// TwinCAT 3 PLC project PLC
// ProgramVersion: 3.1.4023.0
// libraries:
//   Tc2_Standard, * (Beckhoff Automation GmbH)
//   Tc2_System, * (Beckhoff Automation GmbH)
//   Tc2_Utilities, * (Beckhoff Automation GmbH)
//   Tc3_Module, * (Beckhoff Automation GmbH)
//   VisuDialogs, * (System)
//   VisuSymbols,3.5.10.0,System
// project tree:
//   / GlobalTextList.TcGTLO, PlcTask.TcTTO, Visualization Manager.TcVMO (not stored)
//   GVLs/ GVL_Elementy.TcGVL, GVL_Wejscia_IO.TcGVL, GVL_Wyjscia_IO.TcGVL (not stored)
//   POUs/01 - Elementy/Czujnik/ITF/ ITF_Czujnik.TcIO (not stored)
//   POUs/01 - Elementy/Czujnik/POU/ FB_Czujnik_NO.TcPOU (not stored), FB_Czujnik_NC.TcPOU (not stored)
//   POUs/01 - Elementy/Elektrozawór/ITF/ ITF_Elektozawor.TcIO (not stored)
//   POUs/01 - Elementy/Elektrozawór/POU/ FB_Elektrozawor_5na2_1Cewka.TcPOU (not stored), FB_Elektrozawor_5na2_2Cewki.TcPOU (not stored), FB_Elektrozawor_5na3_Odpowietrzony.TcPOU (not stored), FB_Elektrozawor_5na3_Zapowietrzony.TcPOU (not stored)
//   POUs/01 - Elementy/Silownik/DUT/ DUT_SilownikParametry.TcDUT (not stored)
//   POUs/01 - Elementy/Silownik/ITF/ ITF_Silownik.TcIO (not stored)
//   POUs/01 - Elementy/Silownik/POU/ FB_Silownik.TcPOU (not stored), FB_Silownik_Kontola.TcPOU (not stored), FB_Silownik_Kontrola_Komunikacja.TcPOU (not stored)
//   POUs/02 -Przesuwacz Na Silowniku/DUT/ DUT_PrzesuwaczNaSilowniku_Parametry.TcDUT (not stored)
//   POUs/02 -Przesuwacz Na Silowniku/POU/ FB_PrzesuwaczNaSilowniku.TcPOU, FB_PrzesuwaczNaSilowniku_Komunikacja.TcPOU (not stored)
//   POUs/10 - Logowanie błędów/DUT/ DUT_LogowanieBledow_Zapamietanych.TcDUT (not stored), DUT_LogowanieBledow_ZdarzenieOpis.TcDUT (not stored), DUT_LogowanieBledow_Zdarzenie.TcDUT (not stored), DUT_LogowanieBledow_ZdarzenieStan.TcDUT (not stored), DUT_LogowanieBledow_ZdarzenieWyswietlane.TcDUT, DUT_LogowanieBledow_WyswietlanieParametry.TcDUT (not stored)
//   POUs/10 - Logowanie błędów/GVL/ GVL_LogowanieBledow.TcGVL, GVL_LogowanieBledow_Stale.TcGVL
//   POUs/10 - Logowanie błędów/ITF/ ITF_LogowanieBledow_ElementWykonawczy.TcIO (not stored)
//   POUs/10 - Logowanie błędów/POU/ FB_LogowanieBledow.TcPOU, FB_LogowanieBledow_ElementWykonawczy.TcPOU, FB_LogowanieBledow_ElementZlozony.TcPOU
//   POUs/10 - Logowanie błędów/Wizualizacja/ Visu_LogowanieBledow_Tabela.TcVIS
//   POUs/ MAIN.TcPOU
//   VISUs/ Visualization.TcVIS
// real-time tasks:
//   TASK PlcTask: cycle T#10ms, priority 20, ADS port 350

CONFIGURATION PLC
    RESOURCE PLC ON TwinCAT3
        TASK PlcTask(INTERVAL := T#10ms, PRIORITY := 20);
        PROGRAM MAIN WITH PlcTask : MAIN;
    END_RESOURCE
END_CONFIGURATION

// ---- POUs/10 - Logowanie błędów/DUT/DUT_LogowanieBledow_ZdarzenieWyswietlane.TcDUT
TYPE DUT_LogowanieBledow_ZdarzenieWyswietlane :
STRUCT
	sNrKomponentu							: STRING[10];
	sKodBledu								: STRING[10];
	byRodzajZdarzenia						: BYTE;
	sOpis									: STRING;
	dtDataStart								: DT;
	dtDateKoniec							: DT;
	dwKolor									: UDINT;
END_STRUCT
END_TYPE

// ---- GVLs/GVL_Elementy.TcGVL
{attribute 'qualified_only'}
{attribute 'global_init_slot' := '40520'}
VAR_GLOBAL
	fbSilownik								: FB_Silownik_Kontola (		fbCzujnikPozycja0 			:= GVL_Wejscia_IO.bCzujnik0S1, 
																		fbCzujnikPozycjaMax 		:= GVL_Wejscia_IO.bCzujnikMaxS1,
																		fbElektrozawor 				:= GVL_Wyjscia_IO.fbElektrozaworS1);
	fbSilownik1								: FB_Silownik_Kontola (		fbCzujnikPozycja0 			:= GVL_Wejscia_IO.bCzujnik0S2, 
																		fbCzujnikPozycjaMax 		:= GVL_Wejscia_IO.bCzujnikMaxS2,
																		fbElektrozawor 				:= GVL_Wyjscia_IO.fbElektrozaworS2);																
	fbPrzesuwacz							: FB_PrzesuwaczNaSilowniku (bCzujnik0Zabieraka			:= GVL_Wejscia_IO.bCzujnik0Z,
		                                                                bCzujnikMaxZabieraka		:= GVL_Wejscia_IO.bCzujnikMaxZ	,
	                                                                    fbElektrozaworZabieraka		:= GVL_Wyjscia_IO.fbElektrozaworZ,
	                                                                    bCzujnik0Przesuwacza		:= GVL_Wejscia_IO.bCzujnik0P,
	                                                                    bCzujnikMaxPrzesuwacza		:= GVL_Wejscia_IO.bCzujnikMaxP	,
	                                                                    fbElektrozaworPrzesuwacza	:= GVL_Wyjscia_IO.fbElektrozaworP);
END_VAR

// ---- GVLs/GVL_Wejscia_IO.TcGVL
{attribute 'qualified_only'}
{attribute 'global_init_slot' := '40501'}
VAR_GLOBAL
//czujniki siłownik1
	bCzujnik0S1								: FB_Czujnik_NO;
	bCzujnikMaxS1							: FB_Czujnik_NO;
//czujniki siłownika2 
	bCzujnik0S2								: FB_Czujnik_NO;
	bCzujnikMaxS2							: FB_Czujnik_NO;
//czujniki przesuwacza
	bCzujnik0Z								: FB_Czujnik_NO;
	bCzujnikMaxZ							: FB_Czujnik_NO;
	bCzujnik0P								: FB_Czujnik_NO;
	bCzujnikMaxP							: FB_Czujnik_NO;
END_VAR

// ---- POUs/10 - Logowanie błędów/GVL/GVL_LogowanieBledow.TcGVL
{attribute 'qualified_only'}
{attribute 'global_init_slot' := '40550'}
VAR_GLOBAL
	arrElementyWykonawcze 					: ARRAY [1..GVL_LogowanieBledow_Stale.MAX_ILOSC_ELEMENTOW] OF 
																ITF_LogowanieBledow_ElementWykonawczy := [
																	GVL_Elementy.fbSilownik.fbLBKomunikacja, 
																	GVL_Elementy.fbSilownik1.fbLBKomunikacja,
																	GVL_Elementy.fbPrzesuwacz.fbLBKomunikacja];

	fbLoger 								: FB_LogowanieBledow (	tablica := arrElementyWykonawcze,
																	iIloscDodanychElementow := 3);
																	
	
END_VAR
VAR_GLOBAL //PERSISTENT
	arrTablicaZdarzenZapamietancyh			: ARRAY [1..GVL_LogowanieBledow_Stale.MAX_ILOSC_ZDARZEN_ZAPAMIETANYCH] OF DUT_LogowanieBledow_Zapamietanych;																
	
	iIloscZdarzenZapamietanych				: INT;	//ilosc zdarzen ktore wystapiły
END_VAR

// ---- POUs/10 - Logowanie błędów/GVL/GVL_LogowanieBledow_Stale.TcGVL
{attribute 'qualified_only'}
VAR_GLOBAL CONSTANT
	MAX_ILOSC_ELEMENTOW						: INT := 10; //Ilementów głównych
	MAX_ILOSC_ZDARZEN_NA_ELEMENT			: INT := 10;
	MAX_ILOSC_ELEMENTOW_NA_PODZESPOL		: INT := 10;
	MAX_ILOSC_ZDARZEN						: INT := 100;
	MAX_ILOSC_ZDARZEN_DO_WYSWIETLANIA		: INT := 50;
END_VAR

// ---- POUs/MAIN.TcPOU
//==================================================================================================
//								RJM Maszyny sp. z o.o.
//									13.05.2022
//	Program główny sterujący  
// 	v1.0	|| TC v 3.1.4024.29		|| - pierwsza wersja
//==================================================================================================
PROGRAM MAIN
VAR
	bDoPoczatku								: BOOL;
	bDoKonca								: BOOL;
	bNaPoczatku								: BOOL;
	bNaKoncu								: BOOL;
	bWykonajCyklPrzesuwania					: BOOL;
	bWyswietlAlarmy							: BOOL;

END_VAR

(* 	DO ZROBIENIA
	LOGOWANIE BLEDOW
		- poprawić wizualizację logowania błędów nie działają przyciski wyboru rodzaju informacji 
		- id zdarzenia to string nei da się filtrować po id bo nei da się wpisać numerka
		- na maszynie odznaczyc PERSISTENT
		- funkcja czyszczenia tablicy zapamietanych 
	
*)

//--------TESTY FB SILOWNIK
	GVL_Elementy.fbSilownik.Praca ();
	GVL_Elementy.fbPrzesuwacz.Praca ();
	
	IF (bDoPoczatku) THEN
		GVL_Elementy.fbSilownik.PrzesunDoPoczatku	:= TRUE;
		bDoPoczatku							:= FALSE;
	END_IF
	
	IF (bDoKonca) THEN
		GVL_Elementy.fbSilownik.PrzesunDoKonca	:= TRUE;
		bDoKonca							:= FALSE;
	END_IF
	
	bNaPoczatku								:= GVL_Elementy.fbSilownik.NaPoczatku;
	bNaKoncu								:= GVL_Elementy.fbSilownik.NaKoncu;
	
	IF (bWykonajCyklPrzesuwania) THEN
		GVL_Elementy.fbPrzesuwacz.WykonajCyklPrzesuwania	:= TRUE;
		bWykonajCyklPrzesuwania				:= FALSE;
	END_IF
//--------TESTY FB SILOWNIK
//--------LOGER
	GVL_LogowanieBledow.fbLoger (arrZdarzeniaPamietane 		:= GVL_LogowanieBledow.arrTablicaZdarzenZapamietancyh,
								iIloscZdarzenZapamietanych 	:= GVL_LogowanieBledow.iIloscZdarzenZapamietanych,
								bWyswietlanieTablicyAlarmow	:= bWyswietlAlarmy);
//--------LOGER
												
//--------STEROWANIE MASZYNĄ

//--------STEROWANIE MASZYNĄ

END_PROGRAM

// ---- POUs/02 -Przesuwacz Na Silowniku/POU/FB_PrzesuwaczNaSilowniku.TcPOU
//==================================================================================================
//								RJM Maszyny sp. z o.o.
//									13.05.2022
//	Obsluga przesuwacza na siłowniku 
//	Siłownik zabieraka plus siłownik przesuwający 
//	Cykl przesuwania: wysun zabierak -> przesun -> schowaj zabierak -> powrót  
// 	v1.0	|| TC v 3.1.4024.22		|| - pierwsza wersja
//==================================================================================================
FUNCTION_BLOCK FB_PrzesuwaczNaSilowniku
VAR_INPUT
END_VAR
VAR_OUTPUT
END_VAR
VAR
	bCzujnik0Zabieraka						: ITF_Czujnik;
	bCzujnikMaxZabieraka					: ITF_Czujnik;
	fbElektrozaworZabieraka					: ITF_Elektozawor;
	bCzujnik0Przesuwacza					: ITF_Czujnik;
	bCzujnikMaxPrzesuwacza					: ITF_Czujnik;
	fbElektrozaworPrzesuwacza				: ITF_Elektozawor;
	fbZabierak								: FB_Silownik_Kontola (fbCzujnikPozycja0 		:= bCzujnik0Zabieraka, 
																	fbCzujnikPozycjaMax 	:= bCzujnikMaxZabieraka,
																	fbElektrozawor 			:= fbElektrozaworZabieraka);
	fbPrzesuwaczNaped						: FB_Silownik_Kontola (fbCzujnikPozycja0 		:= bCzujnik0Przesuwacza, 
																	fbCzujnikPozycjaMax 	:= bCzujnikMaxPrzesuwacza,
																	fbElektrozawor 			:= fbElektrozaworPrzesuwacza);	
	arrElementyWykonawcze 					: ARRAY [1..10] OF ITF_LogowanieBledow_ElementWykonawczy := 
														[fbZabierak.fbLBKomunikacja, 
														fbPrzesuwaczNaped.fbLBKomunikacja];
	fbLBKomunikacja							: FB_PrzesuwaczNaSilowniku_Komunikacja 
														(arrElementyWykonawcze := arrElementyWykonawcze,
														iIloscPodlementow := 2);
END_VAR

METHOD FB_init : BOOL
VAR_INPUT
	bInitRetains : BOOL; // if TRUE, the retain variables are initialized (warm start / cold start)
	bInCopyCode : BOOL;  // if TRUE, the instance afterwards gets moved into the copy code (online change)
	bCzujnik0Zabieraka						: ITF_Czujnik;
	bCzujnikMaxZabieraka					: ITF_Czujnik;
	fbElektrozaworZabieraka					: ITF_Elektozawor;
	bCzujnik0Przesuwacza					: ITF_Czujnik;
	bCzujnikMaxPrzesuwacza					: ITF_Czujnik;
	fbElektrozaworPrzesuwacza				: ITF_Elektozawor;
END_VAR
THIS^.bCzujnik0Zabieraka					:= bCzujnik0Zabieraka;			     
THIS^.bCzujnikMaxZabieraka					:= bCzujnikMaxZabieraka;		    
THIS^.fbElektrozaworZabieraka				:= fbElektrozaworZabieraka;		 
THIS^.bCzujnik0Przesuwacza					:= bCzujnik0Przesuwacza;		    
THIS^.bCzujnikMaxPrzesuwacza				:= bCzujnikMaxPrzesuwacza;		  
THIS^.fbElektrozaworPrzesuwacza				:= fbElektrozaworPrzesuwacza;

THIS^.fbZabierak.FB_init (FALSE, FALSE, bCzujnik0Zabieraka, bCzujnikMaxZabieraka, fbElektrozaworZabieraka);
THIS^.fbPrzesuwaczNaped.FB_init (FALSE, FALSE, bCzujnik0Przesuwacza, bCzujnikMaxPrzesuwacza, fbElektrozaworPrzesuwacza);
END_METHOD

END_FUNCTION_BLOCK

// ---- POUs/10 - Logowanie błędów/POU/FB_LogowanieBledow.TcPOU
//==================================================================================================
//							RJM MASZYNY SP. Z O>O>
//									05.02.2022
//	Metoda sterujaca logowaniem bledow
// 	v1.0	|| TC v 3.1.4024.22		|| - pierwsza wersja
//==================================================================================================
FUNCTION_BLOCK FB_LogowanieBledow
VAR_INPUT
	arrZdarzeniaPamietane					: REFERENCE TO ARRAY [1..GVL_LogowanieBledow_Stale.MAX_ILOSC_ZDARZEN_ZAPAMIETANYCH] OF DUT_LogowanieBledow_Zapamietanych;
	iIloscZdarzenZapamietanych				: REFERENCE TO INT;
	bWyswietlanieTablicyAlarmow				: BOOL;
END_VAR
VAR_OUTPUT
END_VAR
VAR
	arrTablicaElementowWykonawczych 		: ARRAY [1..GVL_LogowanieBledow_Stale.MAX_ILOSC_ELEMENTOW] OF ITF_LogowanieBledow_ElementWykonawczy;
	iIloscDodanychElementow					: INT;			//ilość dodanych elementow wykonawczych, przypisać w deklaracji
	iIloscDodanychWszystkichZdarzen 		: INT;			//ilosść dodanych zdarzeń globalnie
	iJezykID								: INT := 1045;	//id języka - domyślnie polski
	bwypelnij								: BOOL;			//Wypełnienie tablic - wykonać na początku i po zmianie języka
	bDaneWypelnione							: BOOL := FALSE;//jak true mozna odczytywac stany podzespolow
	iI										: INT;
	iJ										: INT;
	
	arrTablicaDefinicjiZdarzen				: ARRAY [1..GVL_LogowanieBledow_Stale.MAX_ILOSC_ZDARZEN] OF DUT_LogowanieBledow_Zdarzenie;
	arrTablicaDefinicjiZdarzenOpis			: ARRAY [1..GVL_LogowanieBledow_Stale.MAX_ILOSC_ZDARZEN] OF DUT_LogowanieBledow_ZdarzenieOpis;
	arrTablicaDefinicjiZdarzenStan			: ARRAY [1..GVL_LogowanieBledow_Stale.MAX_ILOSC_ZDARZEN] OF DUT_LogowanieBledow_ZdarzenieStan;
	arrTablicaWyswietlana					: ARRAY [1..GVL_LOgowanieBledow_Stale.MAX_ILOSC_ZDARZEN_DO_WYSWIETLANIA] OF DUT_LogowanieBledow_ZdarzenieWyswietlane;
	arrPoczatekZdarzenia					: ARRAY [1..GVL_LogowanieBledow_Stale.MAX_ILOSC_ZDARZEN] OF R_TRIG;
	arrKoniecZdarzenia						: ARRAY [1..GVL_LogowanieBledow_Stale.MAX_ILOSC_ZDARZEN] OF F_TRIG;

	fbLocalSystemTime						: FB_LocalSystemTime;
	stAktualnyCzas							: TIMESTRUCT;				// Aktualny czas sytemowy w formie struktury
	dtAktualnyCzas							: DT;		
	bBladRozmiaruTablicyMozliwychZdarzen	: BOOL;						// Niewlasciwy rozmiar tablicy zdarzen - sprawdz HS_ILOSC_ZDARZEN_PAMIETANYCH
	bReferencjaOK							: BOOL;
	bInicjalizacjaDanychTablicyPamietanych	: BOOL := FALSE;
	tonOdswierzanieTablicyPamieci			: TON;
	tOdswierzenieTablicyPamieci				: TIME := T#100MS;
	bOdswierzanieCiagle						: BOOL;
	tonOdswierzaniaTablicyWyswietlania		: TON;
	tOdswierzaniaTablicyWyswietlania		: TIME := T#200MS;
	stWyswietlanieParametry					: DUT_LogowanieBledow_WyswietlanieParametry;
	bWiecejDanychZapamietanych				: BOOL;	//informacja ze jest wiecej danych zapamietanych niz do wyswietlenia
END_VAR

//Pobranie aktualnego czasu systemu
	fbLocalSystemTime (bEnable:= TRUE, systemTime=> stAktualnyCzas);
	dtAktualnyCzas								:= SYSTEMTIME_TO_DT(stAktualnyCzas);
//Sprawdzenie błędów rozmiaru tablic 
	bBladRozmiaruTablicyMozliwychZdarzen 		:= GVL_LogowanieBledow_Stale.MAX_ILOSC_ZDARZEN < 5 OR
													GVL_LogowanieBledow_Stale.MAX_ILOSC_ZDARZEN > 1000;
//Nie ma błędów pracuj z tablicami
	bReferencjaOK := __ISVALIDREF (arrZdarzeniaPamietane);

	IF (NOT bBladRozmiaruTablicyMozliwychZdarzen AND bReferencjaOK) THEN
	//Inicjalizacja tablicy przy starcie 
		Inicjalizacja ();
	//Wypełnienie tablicy zdarzen dla wszystkich elementow
		IF(bwypelnij) THEN
			WypelnianieTablicyZdarzen ();
		END_IF
	//Aktualizacja tablicy stanów
	//Timer odswiezania
		tonOdswierzanieTablicyPamieci(IN:= NOT tonOdswierzanieTablicyPamieci.Q, PT:= tOdswierzenieTablicyPamieci, Q=> , ET=> );
		IF (bDaneWypelnione AND (bOdswierzanieCiagle OR tonOdswierzanieTablicyPamieci.Q)) THEN
			ObslugaAktywnychZdarzen ();
		END_IF		
	//Odswierzanie tablicy alarmow
		tonOdswierzaniaTablicyWyswietlania(IN:= NOT tonOdswierzaniaTablicyWyswietlania.Q,
											 PT:= tOdswierzaniaTablicyWyswietlania, Q=> , ET=> );		// Timer odswiezania
		IF (bWyswietlanieTablicyAlarmow) THEN
			Wyswietlanie ();
		END_IF
	END_IF

METHOD FB_init : BOOL
VAR_INPUT
	bInitRetains : BOOL; // if TRUE, the retain variables are initialized (warm start / cold start)
	bInCopyCode : BOOL;  // if TRUE, the instance afterwards gets moved into the copy code (online change)
	tablica 								: ARRAY [1..GVL_LogowanieBledow_Stale.MAX_ILOSC_ELEMENTOW] OF ITF_LogowanieBledow_ElementWykonawczy;
	iIloscDodanychElementow					: INT;
END_VAR
THIS^.arrTablicaElementowWykonawczych 								:= tablica;
THIS^.iIloscDodanychElementow				:= iIloscDodanychElementow;
END_METHOD

//==================================================================================================
//							RJM MASZYNY SP. Z O>O>
//									05.02.2022
//	Inicjalizacja tablicy zapamietanych zdarzen
//	Wyszukanie niezakonczonych i konczymy
// 	v1.0	|| TC v 3.1.4024.22		|| - pierwsza wersja
//==================================================================================================
METHOD PRIVATE Inicjalizacja : BOOL
VAR_INPUT
END_VAR
		IF (NOT bInicjalizacjaDanychTablicyPamietanych) THEN
			bInicjalizacjaDanychTablicyPamietanych	:= TRUE;
			FOR iJ := 1 TO iIloscZdarzenZapamietanych DO
				IF (arrZdarzeniaPamietane [iJ].bAktywne) THEN
					arrZdarzeniaPamietane [iJ].bAktywne	:= FALSE;
					//wywolac ZadanieKonie();
				END_IF
			END_FOR
		END_IF
END_METHOD

//==================================================================================================
//							RJM MASZYNY SP. Z O>O>
//									05.02.2022
//	Skanowanie tablicy stanow i po pojawieniu sie aktywnego zdarzenia dodajemy do tablicy pamietanych
//	po zakonczeniu aktywnosci zgloszenia zmieniamy w tablicy pamietanych
// 	v1.0	|| TC v 3.1.4024.22		|| - pierwsza wersja
//==================================================================================================
METHOD PRIVATE ObslugaAktywnychZdarzen : BOOL
VAR_INPUT
END_VAR
	FOR iJ := 1 TO iIloscDodanychElementow DO
		arrTablicaElementowWykonawczych [iJ].ZwrocTabliceStanu (arrTablicaDefinicjiZdarzenStan := arrTablicaDefinicjiZdarzenStan);
	END_FOR
	
	FOR iJ := 1 TO iIloscDodanychWszystkichZdarzen DO
		arrPoczatekZdarzenia [iJ] (CLK := arrTablicaDefinicjiZdarzenStan [iJ].bAktywne);
		IF (arrPoczatekZdarzenia [iJ].Q) THEN
		//dodac nowe zdarzenie do tablicy arrZdarzeniaPamietane
			ZdarzeniePoczatek (iIdZdarzenia 	:= arrTablicaDefinicjiZdarzen [iJ].iIdZdarzenia,
								dtAktualnyCzas 	:= dtAktualnyCzas);
		END_IF
		arrKoniecZdarzenia [iJ] (CLK := arrTablicaDefinicjiZdarzenStan [iJ].bAktywne);
		IF (arrKoniecZdarzenia [iJ].Q) THEN
		//odznaczyc koniec zdarzenia w tablicy arrZdarzeniaPamietane
			ZdarzenieKoniec (iNumerWiersza 		:= ZnajdzZdarzenieWTablicyPamietanychPoID (iIDZdarzenia := arrTablicaDefinicjiZdarzen [iJ].iIdZdarzenia),
								dtAktualnyCzas 	:= dtAktualnyCzas);
		END_IF
	END_FOR
END_METHOD

//==================================================================================================
//							RJM MASZYNY SP. Z O>O>
//									05.02.2022
//	Pobieranie danych zdarzen od podelementow systemu i dopisywanie ich do tablicy zdarzen
// 	v1.0	|| TC v 3.1.4024.22		|| - pierwsza wersja
//==================================================================================================
METHOD PRIVATE WypelnianieTablicyZdarzen : BOOL
VAR_INPUT
END_VAR
	bDaneWypelnione						:= FALSE;
	FOR iI := 1 TO iIloscDodanychElementow DO 
		arrTablicaElementowWykonawczych [iI].ZwrocTabliceDefinicji (	
												arrTablicaDefinicjiZdarzen := arrTablicaDefinicjiZdarzen,
												arrTablicaDefinicjiZdarzenOpis := arrTablicaDefinicjiZdarzenOpis,
												arrTablicaDefinicjiZdarzenStan := arrTablicaDefinicjiZdarzenStan,
												iIdZdarzenia := iIloscDodanychWszystkichZdarzen, 
												iNrPodzespolu := iI, 
												iNrPodelementu := 1,
												iNrElementu := 1, 
												iJezykId := iJezykID);
	END_FOR
	bwypelnij 							:= FALSE;
	bDaneWypelnione						:= TRUE;
END_METHOD

//==================================================================================================
//							RJM MASZYNY SP. Z O>O>
//									05.02.2022
//	Start wypelniania tablicy zdarzen
// 	v1.0	|| TC v 3.1.4024.22		|| - pierwsza wersja
//==================================================================================================
PROPERTY WypelnijTabliceZdarzen : BOOL
SET
bwypelnij									:= WypelnijTabliceZdarzen;
END_SET
END_PROPERTY

METHOD PRIVATE Wyswietlanie : BOOL
VAR_INPUT
END_VAR

VAR
	j										: INT;
	i										: INT;
	bUsunZWyswietlania						: BOOL;
END_VAR
IF (tonOdswierzaniaTablicyWyswietlania.Q) THEN
	MEMSET(ADR(arrTablicaWyswietlana),0,SIZEOF(arrTablicaWyswietlana));
	j										:= 1; //wskaznik wierszy tablicy wyswietlania
	bWiecejDanychZapamietanych				:= FALSE;
	FOR i := 1 TO iIloscZdarzenZapamietanych DO
		bUsunZWyswietlania					:= FALSE;	
		IF (arrZdarzeniaPamietane [i].iIDZdarzenia <> 0) THEN	//sprawdzenie czy w wierszu sa jakies dane
			//Ustawienie filtrow wyswietlania
			bUsunZWyswietlania				:= stWyswietlanieParametry.bFiltrID AND stWyswietlanieParametry.iFiltrID <> arrTablicaDefinicjiZdarzen [arrZdarzeniaPamietane [i].iIDZdarzenia].byRodzajZdarzenia;
//			bUsunZWyswietlania				:= bUsunZWyswietlania OR (stWyswietlanieParametry.bFiltrRodzaj AND stWyswietlanieParametry.byFiltrRodzaj <> arrTablicaDefinicjiZdarzen [arrZdarzeniaPamietane [i].iIDZdarzenia].byRodzajZdarzenia);
			bUsunZWyswietlania				:= bUsunZWyswietlania OR (stWyswietlanieParametry.bFiltrStartOD AND arrZdarzeniaPamietane [i].dtDataStart <= stWyswietlanieParametry.dtFiltrStartOD);
			bUsunZWyswietlania				:= bUsunZWyswietlania OR (stWyswietlanieParametry.bFiltrStartDO AND arrZdarzeniaPamietane [i].dtDataStart >= stWyswietlanieParametry.dtFiltrStartDO);
			bUsunZWyswietlania				:= bUsunZWyswietlania OR (stWyswietlanieParametry.bFiltrKoniecOD AND arrZdarzeniaPamietane [i].dtDataKoniec <= stWyswietlanieParametry.dtFiltrKoniecOD);
			bUsunZWyswietlania				:= bUsunZWyswietlania OR (stWyswietlanieParametry.bFiltrKoniecDO AND arrZdarzeniaPamietane [i].dtDataKoniec >= stWyswietlanieParametry.dtFiltrKoniecDO);
			bUsunZWyswietlania				:= bUsunZWyswietlania OR (stWyswietlanieParametry.bFiltrAktywne AND DT#1970-1-1-0:0:0 <> arrZdarzeniaPamietane[i].dtDataKoniec);
			// Analogicznie dodajemy inne filtry jesli jest taka potrzeba
			// Jesli element nie zostal usuniety przez filtr to dodajemy go do tablicy alarmow wyswietlanych
			IF (NOT bUsunZWyswietlania) THEN
				arrTablicaWyswietlana [j].sNrKomponentu	:= arrTablicaDefinicjiZdarzen [i].sNrKomponentu;
				arrTablicaWyswietlana [j].byRodzajZdarzenia	:= arrTablicaDefinicjiZdarzen [i].byRodzajZdarzenia;
 				arrTablicaWyswietlana [j].sOpis			:= arrTablicaDefinicjiZdarzenOpis [i].sOpis;
				arrTablicaWyswietlana [j].sKodBledu		:= arrTablicaDefinicjiZdarzen [i].sKodBledu;
				arrTablicaWyswietlana [j].dtDataStart	:= arrZdarzeniaPamietane [i].dtDataStart;
				arrTablicaWyswietlana [j].dtDataKoniec	:= arrZdarzeniaPamietane [i].dtDataKoniec;
				CASE arrTablicaWyswietlana [j].byRodzajZdarzenia OF
					1	: arrTablicaWyswietlana [j].dwKolor	:= 16#FFFF0000;	// blad 		- czerwony
					2	: arrTablicaWyswietlana [j].dwKolor	:= 16#FFFFFF00;	// ostzrezenie 	- zolty
					3	: arrTablicaWyswietlana [j].dwKolor	:= 16#FFFFFFFF;	// wiadomosc 	- bialy
					4	: arrTablicaWyswietlana [j].dwKolor	:= 16#FF0000FF; // safety 		- niebieski
				END_CASE
				j := j + 1;
			END_IF
		END_IF
		IF (j > GVL_LogowanieBledow_Stale.MAX_ILOSC_ZDARZEN_DO_WYSWIETLANIA) THEN
			bWiecejDanychZapamietanych		:= TRUE;
			EXIT;
		END_IF
	END_FOR
END_IF
END_METHOD

//==================================================================================================
//							RJM MASZYNY SP. Z O>O>
//									05.02.2022
//	Zdarzenie przestalo byc aktywne zmien dane
// 	v1.0	|| TC v 3.1.4024.22		|| - pierwsza wersja
//==================================================================================================
METHOD PRIVATE ZdarzenieKoniec : BOOL
VAR_INPUT
	iNumerWiersza							: INT;	//numer wiersza dla konkretnego IDzdarzenia
	dtAktualnyCzas							: DT;
END_VAR
arrZdarzeniaPamietane [iNumerWiersza].dtDataKoniec	:= dtAktualnyCzas;
arrZdarzeniaPamietane [iNumerWiersza].bAktywne		:= FALSE;
END_METHOD

//==================================================================================================
//							RJM MASZYNY SP. Z O>O>
//									05.02.2022
//	Dodanie nowego aktywnego zdarzenia do tablicy pamietanych
// 	v1.0	|| TC v 3.1.4024.22		|| - pierwsza wersja
//==================================================================================================
METHOD PRIVATE ZdarzeniePoczatek : BOOL
VAR_INPUT
	iIdZdarzenia							: INT;
	dtAktualnyCzas							: DT;
END_VAR
VAR
	i										: INT;
END_VAR
iIloscZdarzenZapamietanych					:= iIloscZdarzenZapamietanych + 1;
// Przesun elemety tablicy
FOR i := 0 TO iIloscZdarzenZapamietanych - 2 DO
	arrZdarzeniaPamietane [iIloscZdarzenZapamietanych - i]	:= arrZdarzeniaPamietane [iIloscZdarzenZapamietanych - i - 1];
END_FOR

// Dodaj nowy
//arrZdarzeniaPamietane [1].dwIDZdarzenia		:= stZdarzenie.dwIDZdarzenia;
arrZdarzeniaPamietane [1].iIDZdarzenia		:= iIDZdarzenia;
arrZdarzeniaPamietane [1].dtDataStart		:= dtAktualnyCzas;
arrZdarzeniaPamietane [1].dtDataKoniec		:= DT#1970-1-1-0:0:0;
arrZdarzeniaPamietane [1].bAktywne			:= TRUE;
END_METHOD

//==================================================================================================
//							RJM MASZYNY SP. Z O>O>
//									05.02.2022
//	Zwraca numer wiersza w tabeli pamieci z podanym idzdarzenia
// 	v1.0	|| TC v 3.1.4024.22		|| - pierwsza wersja
//==================================================================================================

METHOD PROTECTED ZnajdzZdarzenieWTablicyPamietanychPoID : INT
VAR_INPUT
	iIDZdarzenia							: INT;
END_VAR
VAR 
	i										: INT;
END_VAR
FOR i := 1 TO iIloscZdarzenZapamietanych DO
	IF (arrZdarzeniaPamietane [i].iIDZdarzenia = iIDZdarzenia) THEN
		ZnajdzZdarzenieWTablicyPamietanychPoID	:= i;
		EXIT;
	END_IF
END_FOR
END_METHOD

END_FUNCTION_BLOCK

// ---- POUs/10 - Logowanie błędów/POU/FB_LogowanieBledow_ElementWykonawczy.TcPOU
//==================================================================================================
//								RJM Maszyny sp. z o.o.
//									14.06.2022
//	FB posredniczący pomiędzy FB a logerem alarmów  
// 	v1.0	|| TC v 3.1.4024.22		|| - pierwsza wersja
//==================================================================================================
FUNCTION_BLOCK FB_LogowanieBledow_ElementWykonawczy IMPLEMENTS ITF_LogowanieBledow_ElementWykonawczy
VAR_INPUT
END_VAR
VAR_OUTPUT
END_VAR
VAR
	iStartId								: INT := 0;	//numer poczatkowy dla podzespolu
	arrTablicaStanow						: ARRAY [1..10] OF BOOL;
END_VAR

//==================================================================================================
//								RJM Maszyny sp. z o.o.
//									14.06.2022
//	Metoda do rozszerzenia z opisem alarmów po niemiecku  
// 	v1.0	|| TC v 3.1.4024.22		|| - pierwsza wersja
//==================================================================================================
METHOD DefinicjaTabeliZdarzen_1031_Niemiecki : BOOL
VAR_INPUT
	arrTablicaDefinicjiZdarzenOpis			: REFERENCE TO ARRAY [1..GVL_LogowanieBledow_Stale.MAX_ILOSC_ZDARZEN] OF DUT_LogowanieBledow_ZdarzenieOpis;

END_VAR
END_METHOD

//==================================================================================================
//								RJM Maszyny sp. z o.o.
//									14.06.2022
//	Metoda do rozszerzenia z opisem alarmów po andgielsku  
// 	v1.0	|| TC v 3.1.4024.22		|| - pierwsza wersja
//==================================================================================================
METHOD DefinicjaTabeliZdarzen_1033_Angielski : BOOL
VAR_INPUT
	arrTablicaDefinicjiZdarzenOpis			: REFERENCE TO ARRAY [1..GVL_LogowanieBledow_Stale.MAX_ILOSC_ZDARZEN] OF DUT_LogowanieBledow_ZdarzenieOpis;

END_VAR
END_METHOD

//==================================================================================================
//								RJM Maszyny sp. z o.o.
//									14.06.2022
//	Metoda do rozszerzenia z opisem alarmów po polsku
// 	v1.0	|| TC v 3.1.4024.22		|| - pierwsza wersja
//==================================================================================================
METHOD DefinicjaTabeliZdarzen_1045_Polski : BOOL
VAR_INPUT
	arrTablicaDefinicjiZdarzenOpis			: REFERENCE TO ARRAY [1..GVL_LogowanieBledow_Stale.MAX_ILOSC_ZDARZEN] OF DUT_LogowanieBledow_ZdarzenieOpis;

END_VAR
END_METHOD

//==================================================================================================
//								RJM Maszyny sp. z o.o.
//									14.06.2022
//	Metoda do rozszerzenia wypełniająca niezmienne dane tablic  
// 	v1.0	|| TC v 3.1.4024.22		|| - pierwsza wersja
//==================================================================================================
METHOD DefinicjaTabeliZdarzen_Ogolna : BOOL
VAR_INPUT
	arrTablicaDefinicjiZdarzen				: REFERENCE TO ARRAY [1..GVL_LogowanieBledow_Stale.MAX_ILOSC_ZDARZEN] OF DUT_LogowanieBledow_Zdarzenie;
	arrTablicaDefinicjiZdarzenOpis			: REFERENCE TO ARRAY [1..GVL_LogowanieBledow_Stale.MAX_ILOSC_ZDARZEN] OF DUT_LogowanieBledow_ZdarzenieOpis;
	arrTablicaDefinicjiZdarzenStan			: REFERENCE TO ARRAY [1..GVL_LogowanieBledow_Stale.MAX_ILOSC_ZDARZEN] OF DUT_LogowanieBledow_ZdarzenieStan;

	iIdZdarzenia							: REFERENCE TO INT;
	iNrPodzespolu							: INT := 0;
	iNrPodelementu							: INT := 0;
	iNrElementu								: INT := 0;
END_VAR
END_METHOD

//==================================================================================================
//								RJM Maszyny sp. z o.o.
//									14.06.2022
//	Metoda składa numer podzespołu z podanych zmiennych 
// 	v1.0	|| TC v 3.1.4024.22		|| - pierwsza wersja
//==================================================================================================
METHOD GenerujNrKomponentu : STRING
VAR_INPUT
	iNrPodzespolu							: INT := 0;
	iNrPodelementu							: INT := 0;
	iNrElementu								: INT := 0;
END_VAR
VAR
	sKod									: STRING;
END_VAR
sKod										:= concat (TO_STRING (iNrPodzespolu*100), '-');
sKod										:= concat (sKod, TO_STRING (iNrPodelementu*10));
sKod										:= concat (sKod, '-');
sKod										:= concat (sKod, TO_STRING (iNrElementu));

GenerujNrKomponentu							:= sKod;
END_METHOD

//==================================================================================================
//								RJM Maszyny sp. z o.o.
//									14.06.2022
//	Przypisanie odpowiedniego stonu w odpowienim miejscu w tabeli potrzebne do aktualizacji stanow alarmow
// 	v1.0	|| TC v 3.1.4024.22		|| - pierwsza wersja
//==================================================================================================
METHOD UstawStan : BOOL
VAR_INPUT
	iId										: INT;
	bStan									: BOOL;
END_VAR
arrTablicaStanow [iId]					:= bStan;
END_METHOD

//==================================================================================================
//								RJM Maszyny sp. z o.o.
//									14.06.2022
//	Metoda zwraca definicje alarmow dla elementów wykonawczych
// 	v1.0	|| TC v 3.1.4024.22		|| - pierwsza wersja
//==================================================================================================
METHOD ZwrocTabliceDefinicji : BOOL
VAR_INPUT
	arrTablicaDefinicjiZdarzen				: REFERENCE TO ARRAY [1..GVL_LogowanieBledow_Stale.MAX_ILOSC_ZDARZEN] OF DUT_LogowanieBledow_Zdarzenie;
	arrTablicaDefinicjiZdarzenOpis			: REFERENCE TO ARRAY [1..GVL_LogowanieBledow_Stale.MAX_ILOSC_ZDARZEN] OF DUT_LogowanieBledow_ZdarzenieOpis;
	arrTablicaDefinicjiZdarzenStan			: REFERENCE TO ARRAY [1..GVL_LogowanieBledow_Stale.MAX_ILOSC_ZDARZEN] OF DUT_LogowanieBledow_ZdarzenieStan;
	
	iIdZdarzenia							: REFERENCE TO INT;
	iNrPodzespolu							: INT;
	iNrPodelementu							: INT;
	iNrElementu								: INT;
	iJezykId								: INT;
END_VAR
	IF (iStartId = 0) THEN
		iStartId							:= iIdZdarzenia+1;
		DefinicjaTabeliZdarzen_Ogolna (	arrTablicaDefinicjiZdarzen 		:= arrTablicaDefinicjiZdarzen,
										arrTablicaDefinicjiZdarzenOpis 	:= arrTablicaDefinicjiZdarzenOpis,
										arrTablicaDefinicjiZdarzenStan 	:= arrTablicaDefinicjiZdarzenStan,
										iIdZdarzenia 					:= iIdZdarzenia,
										iNrPodzespolu 					:= iNrPodzespolu,
										iNrPodelementu 					:= iNrPodelementu,
										iNrElementu						:= iNrElementu);
	END_IF
	
	CASE iJezykId OF
		1031	:	//niemiecki
			DefinicjaTabeliZdarzen_1031_Niemiecki (arrTablicaDefinicjiZdarzenOpis 	:= arrTablicaDefinicjiZdarzenOpis);
		1033	:	//angielski
			DefinicjaTabeliZdarzen_1033_Angielski (arrTablicaDefinicjiZdarzenOpis 	:= arrTablicaDefinicjiZdarzenOpis);
		1045	:	//polski
			DefinicjaTabeliZdarzen_1045_Polski (arrTablicaDefinicjiZdarzenOpis 	:= arrTablicaDefinicjiZdarzenOpis);
		ELSE		//domyslny polski
			DefinicjaTabeliZdarzen_1045_Polski (arrTablicaDefinicjiZdarzenOpis 	:= arrTablicaDefinicjiZdarzenOpis);		
	END_CASE
	
//	ZwrocTabeleZdarzen						REF= arrZdarzeniaDefinicja;
END_METHOD

//==================================================================================================
//								RJM Maszyny sp. z o.o.
//									14.06.2022
//	Metoda zwraca tablice stanow elementu wykonwaczego  
// 	v1.0	|| TC v 3.1.4024.22		|| - pierwsza wersja
//==================================================================================================
METHOD ZwrocTabliceStanu : BOOL
VAR_INPUT
	arrTablicaDefinicjiZdarzenStan			: REFERENCE TO ARRAY [1..GVL_LogowanieBledow_Stale.MAX_ILOSC_ZDARZEN] OF DUT_LogowanieBledow_ZdarzenieStan;
END_VAR

VAR
	iI: INT;
END_VAR
FOR iI := 1 TO 10 DO
	arrTablicaDefinicjiZdarzenStan [iStartId + iI -1].bAktywne := arrTablicaStanow [iI];
END_FOR
END_METHOD

END_FUNCTION_BLOCK

// ---- POUs/10 - Logowanie błędów/POU/FB_LogowanieBledow_ElementZlozony.TcPOU
//==================================================================================================
//								RJM Maszyny sp. z o.o.
//									14.06.2022
//	FB posredniczący pomiędzy FB a logerem alarmów  rozszerzenie dla elementów złożonych
// 	v1.0	|| TC v 3.1.4024.22		|| - pierwsza wersja
//==================================================================================================
FUNCTION_BLOCK FB_LogowanieBledow_ElementZlozony EXTENDS FB_LogowanieBledow_ElementWykonawczy
VAR_INPUT
	
END_VAR
VAR_OUTPUT
END_VAR
VAR
	arrElementyWykonawcze 					: ARRAY [1..10] OF ITF_LogowanieBledow_ElementWykonawczy;
	iIloscPodlementow						: INT;
END_VAR

METHOD DefinicjaTabeliZdarzen_1031_Niemiecki : BOOL
VAR_INPUT
	arrTablicaDefinicjiZdarzenOpis			: REFERENCE TO ARRAY [1..GVL_LogowanieBledow_Stale.MAX_ILOSC_ZDARZEN] OF DUT_LogowanieBledow_ZdarzenieOpis;

END_VAR
END_METHOD

METHOD DefinicjaTabeliZdarzen_1033_Angielski : BOOL
VAR_INPUT
	arrTablicaDefinicjiZdarzenOpis			: REFERENCE TO ARRAY [1..GVL_LogowanieBledow_Stale.MAX_ILOSC_ZDARZEN] OF DUT_LogowanieBledow_ZdarzenieOpis;

END_VAR
END_METHOD

METHOD DefinicjaTabeliZdarzen_1045_Polski : BOOL
VAR_INPUT
	arrTablicaDefinicjiZdarzenOpis			: REFERENCE TO ARRAY [1..GVL_LogowanieBledow_Stale.MAX_ILOSC_ZDARZEN] OF DUT_LogowanieBledow_ZdarzenieOpis;

END_VAR
END_METHOD

METHOD DefinicjaTabeliZdarzen_Ogolna : BOOL
VAR_INPUT
	arrTablicaDefinicjiZdarzen				: REFERENCE TO ARRAY [1..GVL_LogowanieBledow_Stale.MAX_ILOSC_ZDARZEN] OF DUT_LogowanieBledow_Zdarzenie;
	arrTablicaDefinicjiZdarzenOpis			: REFERENCE TO ARRAY [1..GVL_LogowanieBledow_Stale.MAX_ILOSC_ZDARZEN] OF DUT_LogowanieBledow_ZdarzenieOpis;
	arrTablicaDefinicjiZdarzenStan			: REFERENCE TO ARRAY [1..GVL_LogowanieBledow_Stale.MAX_ILOSC_ZDARZEN] OF DUT_LogowanieBledow_ZdarzenieStan;

	iIdZdarzenia							: REFERENCE TO INT;
	iNrPodzespolu							: INT := 0;
	iNrPodelementu							: INT := 0;
	iNrElementu								: INT := 0;
END_VAR
END_METHOD

METHOD FB_init : BOOL
VAR_INPUT
	bInitRetains : BOOL; // if TRUE, the retain variables are initialized (warm start / cold start)
	bInCopyCode : BOOL;  // if TRUE, the instance afterwards gets moved into the copy code (online change)
	arrElementyWykonawcze 					: ARRAY [1..10] OF ITF_LogowanieBledow_ElementWykonawczy;
	iIloscPodlementow						: INT;
END_VAR
THIS^.arrElementyWykonawcze					:= arrElementyWykonawcze;
THIS^.iIloscPodlementow						:= iIloscPodlementow;
END_METHOD

METHOD ZwrocTabliceDefinicji : BOOL
VAR_INPUT
	arrTablicaDefinicjiZdarzen				: REFERENCE TO ARRAY [1..GVL_LogowanieBledow_Stale.MAX_ILOSC_ZDARZEN] OF DUT_LogowanieBledow_Zdarzenie;
	arrTablicaDefinicjiZdarzenOpis			: REFERENCE TO ARRAY [1..GVL_LogowanieBledow_Stale.MAX_ILOSC_ZDARZEN] OF DUT_LogowanieBledow_ZdarzenieOpis;
	arrTablicaDefinicjiZdarzenStan			: REFERENCE TO ARRAY [1..GVL_LogowanieBledow_Stale.MAX_ILOSC_ZDARZEN] OF DUT_LogowanieBledow_ZdarzenieStan;
	
	iIdZdarzenia							: REFERENCE TO INT;
	iNrPodzespolu							: INT;
	iNrPodelementu							: INT;
	iNrElementu								: INT;
	iJezykId								: INT;
END_VAR
VAR
	iI: INT;
END_VAR
//Zwrócenie definicji zdarzen dla głównego elementu 
SUPER^.ZwrocTabliceDefinicji (	arrTablicaDefinicjiZdarzen := arrTablicaDefinicjiZdarzen,
								arrTablicaDefinicjiZdarzenOpis := arrTablicaDefinicjiZdarzenOpis,
								arrTablicaDefinicjiZdarzenStan := arrTablicaDefinicjiZdarzenStan,
								iIdZdarzenia := iIdZdarzenia,
								iNrPodzespolu := iNrPodzespolu, 
								iNrPodelementu := iNrPodelementu,
								iNrElementu := 1, 
								iJezykId := iJezykID);
//zwrócenie tablicy definicji dla podelementów

	FOR iI := 1 TO iIloscPodlementow DO 


//		IF (__ISVALIDREF (arrElementyWykonawcze [iI])) THEN
			arrElementyWykonawcze [iI].ZwrocTabliceDefinicji (	arrTablicaDefinicjiZdarzen := arrTablicaDefinicjiZdarzen,
																arrTablicaDefinicjiZdarzenOpis := arrTablicaDefinicjiZdarzenOpis,
																arrTablicaDefinicjiZdarzenStan := arrTablicaDefinicjiZdarzenStan,
																iIdZdarzenia := iIdZdarzenia, 
																iNrPodzespolu := iNrPodzespolu, 
																iNrPodelementu := iNrPodelementu,
																iNrElementu := iI+1, 
																iJezykId := iJezykID);
//iIdZdarzenia := itest, 
//													iNrPodzespolu := iIdZdarzenia, iNrPodelementu := 1,
//													iNrElementu := 1, iJezykId := iJezykID);
//		ELSE 
//			EXIT;
//		END_IF
	END_FOR
END_METHOD

METHOD ZwrocTabliceStanu : BOOL
VAR_INPUT
	arrTablicaDefinicjiZdarzenStan			: REFERENCE TO ARRAY [1..GVL_LogowanieBledow_Stale.MAX_ILOSC_ZDARZEN] OF DUT_LogowanieBledow_ZdarzenieStan;
END_VAR

VAR
	iI										: INT;
	iJ										: INT;
END_VAR
SUPER^.ZwrocTabliceStanu (arrTablicaDefinicjiZdarzenStan := arrTablicaDefinicjiZdarzenStan);

FOR iJ := 1 TO iIloscPodlementow DO
	arrElementyWykonawcze [iJ].ZwrocTabliceStanu (arrTablicaDefinicjiZdarzenStan := arrTablicaDefinicjiZdarzenStan);
END_FOR
END_METHOD

END_FUNCTION_BLOCK

// ---- GlobalTextList.TcGTLO
TEXTLIST GlobalTextList
  22 = '%s'
  977 = 'Abort'
  836 = 'Bezpieczeństwo'
  340 = 'Błędy'
  0 = 'Clear'
  274 = 'Czas koniec do'
  206 = 'Czas koniec od'
  253 = 'Czas start do'
  809 = 'Czas start od'
  595 = 'Data koniec'
  676 = 'Data start'
  609 = 'Grupa \nwiadomości'
  936 = 'Hold'
  324 = 'ID'
  917 = 'Kod'
  998 = 'Nr Elem.'
  700 = 'Opis'
  516 = 'Ostrzerzenia'
  414 = 'R'
  573 = 'Reset'
  125 = 'Start'
  387 = 'Stop'
  986 = 'Suspend'
  892 = 'Tryb automatyczny'
  740 = 'Tryb reczny'
  916 = 'Tylko aktywne'
  974 = 'Un-hold'
  152 = 'Un-Suspend'
  528 = 'Wiadomości'
END_TEXTLIST

// ---- POUs/10 - Logowanie błędów/Wizualizacja/Visu_LogowanieBledow_Tabela.TcVIS
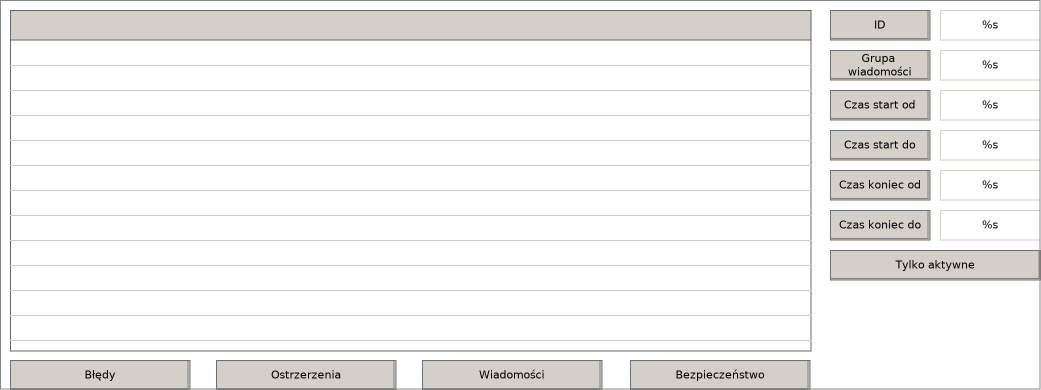
VISUALIZATION Visu_LogowanieBledow_Tabela  // 1041x390
VAR_IN_OUT
	stParametry								: DUT_LogowanieBledow_WyswietlanieParametry;
END_VAR
    Table (10,10 801x341), data array: GVL_LogowanieBledow.fbLoger.arrTablicaWyswietlana
        p3854506369: GVL_LogowanieBledow.fbLoger.arrTablicaWyswietlana[INDEX].sNrKomponentu
        p1892666644: GVL_LogowanieBledow.fbLoger.arrTablicaWyswietlana[INDEX].sKodBledu
        p338671338: GVL_LogowanieBledow.fbLoger.arrTablicaWyswietlana[INDEX].byRodzajZdarzenia
        p2170511999: GVL_LogowanieBledow.fbLoger.arrTablicaWyswietlana[INDEX].sOpis
        p3723444502: GVL_LogowanieBledow.fbLoger.arrTablicaWyswietlana[INDEX].dtDataStart
        p1218418051: GVL_LogowanieBledow.fbLoger.arrTablicaWyswietlana[INDEX].dtDataKoniec
        p746581629: GVL_LogowanieBledow.fbLoger.arrTablicaWyswietlana[INDEX].dwKolor
        p2232123230: Nr Elem.
        p2237128397: Data start
        p505689113: Data koniec
    Button (830,10 100x30), "ID", colour toggle: stParametry.bFiltrID
        toggle stParametry.bFiltrID
    Button (830,50 100x30), "Grupa wiadomości", colour toggle: stParametry.bFiltrRodzaj
        toggle stParametry.bFiltrRodzaj
    Button (830,90 100x30), "Czas start od", colour toggle: stParametry.bFiltrStartOD
        toggle stParametry.bFiltrStartOD
    Button (830,130 100x30), "Czas start do", colour toggle: stParametry.bFiltrStartDO
        toggle stParametry.bFiltrStartDO
    Button (830,170 100x30), "Czas koniec od", colour toggle: stParametry.bFiltrKoniecOD
        toggle stParametry.bFiltrKoniecOD
    Button (830,210 100x30), "Czas koniec do", colour toggle: stParametry.bFiltrKoniecDO
        toggle stParametry.bFiltrKoniecDO
    Button (830,250 211x30), "Tylko aktywne", colour toggle: stParametry.bFiltrAktywne
        toggle stParametry.bFiltrAktywne
    Textfield (940,10 100x30), "%s", text variable: stParametry.iFiltrID
        OnMouseDown: write the text variable via VisuDialogs.Numpad
    Textfield (940,50 100x30), "%s", text variable: stParametry.byFiltrRodzaj
        OnMouseDown: write the text variable via VisuDialogs.Numpad
    Textfield (940,90 100x30), "%s", text variable: stParametry.dtFiltrStartOD
        OnMouseDown: write the text variable via Edit
    Textfield (940,130 100x30), "%s", text variable: stParametry.dtFiltrStartDO
        OnMouseDown: write the text variable via Edit
    Textfield (940,170 100x30), "%s", text variable: stParametry.dtFiltrKoniecOD
        OnMouseDown: write the text variable via Edit
    Textfield (940,210 100x30), "%s", text variable: stParametry.dtFiltrKoniecDO
        OnMouseDown: write the text variable via Edit
    Button (10,360 180x30), "Błędy", colour toggle: stParametry.bFiltrRodzaj and stParametry.byFiltrRodzaj = 1
        OnMouseDown: execute {
            IF (NOT stParametry.bFiltrRodzaj) THEN
            	stParametry.bFiltrRodzaj := TRUE;
            	stParametry.byFiltrRodzaj := 1;
            ELSE
            	stParametry.bFiltrRodzaj := FALSE;
            END_IF
        }
    Button (216,360 180x30), "Ostrzerzenia", colour toggle: stParametry.bFiltrRodzaj and stParametry.byFiltrRodzaj = 2
        OnMouseDown: execute {
            IF (NOT stParametry.bFiltrRodzaj) THEN
            	stParametry.bFiltrRodzaj := TRUE;
            	stParametry.byFiltrRodzaj := 2;
            ELSE
            	stParametry.bFiltrRodzaj := FALSE;
            END_IF
        }
    Button (422,360 180x30), "Wiadomości", colour toggle: stParametry.bFiltrRodzaj and stParametry.byFiltrRodzaj = 3
        OnMouseDown: execute {
            IF (NOT stParametry.bFiltrRodzaj) THEN
            	stParametry.bFiltrRodzaj := TRUE;
            	stParametry.byFiltrRodzaj := 3;
            ELSE
            	stParametry.bFiltrRodzaj := FALSE;
            END_IF
        }
    Button (630,360 180x30), "Bezpieczeństwo", colour toggle: stParametry.bFiltrRodzaj and stParametry.byFiltrRodzaj = 4
        OnMouseDown: execute {
            IF (NOT stParametry.bFiltrRodzaj) THEN
            	stParametry.bFiltrRodzaj := TRUE;
            	stParametry.byFiltrRodzaj := 4;
            ELSE
            	stParametry.bFiltrRodzaj := FALSE;
            END_IF
        }
END_VISUALIZATION

// ---- VISUs/Visualization.TcVIS
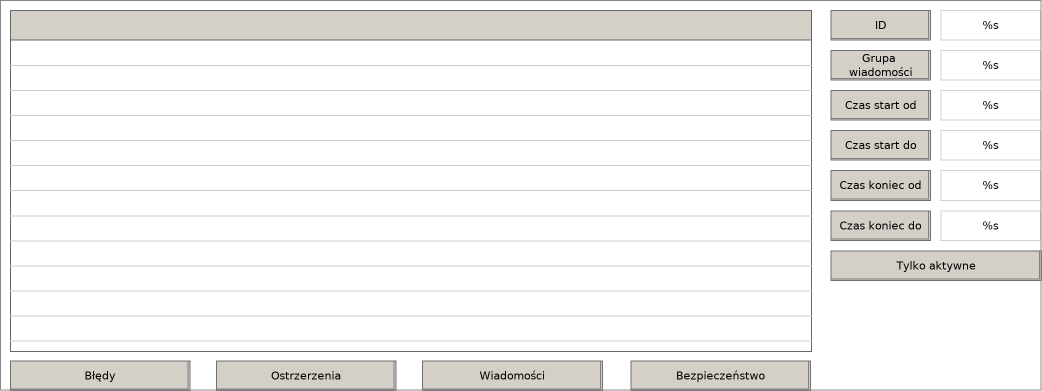
VISUALIZATION Visualization  // 1042x391
    Frame (0,0 1042x391)
        shows Visu_LogowanieBledow_Tabela(stParametry := GVL_LogowanieBledow.fbLoger.stWyswietlanieParametry)
END_VISUALIZATION
